{attribute 'qualified_only'}
VAR_GLOBAL
	// Safety Error Condition
	Error		AT%I*:	BOOL;
	// Run/Stop Safety
	Run			AT%Q*:	BOOL;
	// Restart Safety
	Restart		AT%Q*:	BOOL;
	// Error Acknowledgement 
	ErrAck		AT%Q*:	BOOL;
	// Stop signal coming from Safety
	Stop		AT%I*:	BOOL;
	// state variable
	State		AT%I*:	USINT;
END_VAR

(* stored: Version 1.1.0.1, ProductVersion 3.1.4024.12
   GVL GVL_Safety: Id {53515296-dd36-485f-b9b3-71a8a885417c} *)
